TYPE "PPrf_CoilHandlig"
VERSION : 0.1
// Block: PPrf_CoilHandlig
   STRUCT
      MaterialFeeding : PPrf_CoilHandling_MaterialFeeding;
      WeldingCycle : PPrf_CoilHandling_WeldingCycle;
   END_STRUCT;

END_TYPE
